// TIA Portal V17 export
// export: Created 2023-12-22T15:03:15.3902002Z, ExportSetting WithDefaults, DisplayName Totally Integrated Automation Portal, DisplayVersion V17, DisplayName TIA Portal Openness, DisplayVersion V17, DisplayName TIA Portal Version Control Interface, DisplayVersion V17, DisplayName STEP 7 Professional, DisplayVersion V17, DisplayName STEP 7 Safety, DisplayVersion V17, DisplayName WinCC Advanced, DisplayVersion V17
DATA_BLOCK "KP_3_DB"   // DB523
VERSION : 0.1
// stored: AutoNumber false, DBAccessibleFromOPCUA true, DBAccessibleFromWebserver true, InstanceOfName KP_3, InstanceOfType FB
"KP_3"
   // VAR
   //    limit { S7_SetPoint := 'True'} : Int;
   //    load : Int;
   //    load_last : Int;
   //    KP { S7_SetPoint := 'True'} : Array[0..10] of "DRV_AUMA";
   //    load_ok { S7_SetPoint := 'True'} : Bool;
   // END_VAR
BEGIN
END_DATA_BLOCK
